   A_23_A800Z1.InMonFalse := FALSE;
   A_23_A800Z1.InPreAlarmTrue := FALSE;
   A_23_A800Z1.InPreAlarmFalse := FALSE;
   A_23_A800Z1.InStopTrueTime := FALSE;
   A_23_A800Z1.InStopFalseTime := FALSE;
   A_23_A800Z1.InpTrue := FALSE;
   A_23_A800Z1.InpFaultDev := FALSE;
   A_23_A800Z1.CmdRstTrueTime := FALSE;
   A_23_A800Z1.CmdRstFalseTime := FALSE;
   A_23_A800Z1.CmdRunTimeoutTime := FALSE;
   A_23_A800Z1.CmdFaultReset := FALSE;
   A_23_A800Z1.InLocal := FALSE;
   A_23_A800Z1.spare0305 := FALSE;
   A_23_A800Z1.InReport := FALSE;
   A_23_A800Z1.OutTimeoutTime := FALSE;
   A_23_A800Z1.InHWStop := FALSE;
   A_23_A800Z1.InDPFault := FALSE;
   A_23_A800Z1.OutPreAlarmTrue := FALSE;
   A_23_A800Z1.OutPreAlarmFalse := FALSE;
   A_23_A800Z1.OutFlagPos := FALSE;
   A_23_A800Z1.OutFlagNeg := FALSE;
   A_23_A800Z1.OutpFaultReset := FALSE;
   A_23_A800Z1.OutTrue := FALSE;
   A_23_A800Z1.StFalse := FALSE;
   A_23_A800Z1.StCtoTrue := FALSE;
   A_23_A800Z1.StTrue := FALSE;
   A_23_A800Z1.StCtoFalse := FALSE;
   A_23_A800Z1.StFault := FALSE;
   A_23_A800Z1.OutAlarmNrLog := 0;
   A_23_A800Z1.Par.ParObjectNo := 0;
   A_23_A800Z1.Par.ParMsgType := 0;
   A_23_A800Z1.Par.ParHornCode := 0;
   A_23_A800Z1.Par.ParLogOff := FALSE;
   A_23_A800Z1.Par.spare0401 := FALSE;
   A_23_A800Z1.Par.Par2WorkingCond := FALSE;
   A_23_A800Z1.Par.ParFaultRetry := FALSE;
   A_23_A800Z1.Par.ParBinLevel := FALSE;
   A_23_A800Z1.Par.ParDelayChange := 0;
   A_23_A800Z1.Par.ParDelayTrue := 0;
   A_23_A800Z1.Par.ParDelayFalse := 0;
   A_23_A800Z1.Par.ParTimeoutTrue := 0;
   A_23_A800Z1.Par.ParTimeoutFalse := 0;
   A_23_A800Z1.Par.OutMonTime := 0;
   A_23_A800Z1.Par.OutTransitionTime := 0;
   A_23_A800Z1.Par.OutMonTrue := FALSE;
   A_23_A800Z1.Par.OutMonFalse := FALSE;
   A_23_A800Z1.Par.OutFlagFaultDev := FALSE;
   A_23_A800Z1.Par.OutDelayTime := 0;
//Parameter =A-23-A106Z1 : EMERGENCY STOP FROM +C24
      #A_23_A106Z1.Par.ParObjectNo                             :=735;
      #A_23_A106Z1.Par.ParMsgType                              :=7171;
      #A_23_A106Z1.Par.ParHornCode                             :=2;
      #A_23_A106Z1.Par.ParDelayChange                          :=0;
      #A_23_A106Z1.Par.ParDelayTrue                            :=10;
      #A_23_A106Z1.Par.ParDelayFalse                           :=0;
      #A_23_A106Z1.Par.ParTimeoutTrue                          :=0;
      #A_23_A106Z1.Par.ParTimeoutFalse                         :=0;
      #A_23_A106Z1.Par.ParLogOff                               :=False;
      #A_23_A106Z1.Par.Par2WorkingCond                         :=False;
      #A_23_A106Z1.Par.ParFaultRetry                           :=False;
      #A_23_A106Z1.Par.ParBinLevel                             :=False;
//
//
END_DATA_BLOCK

